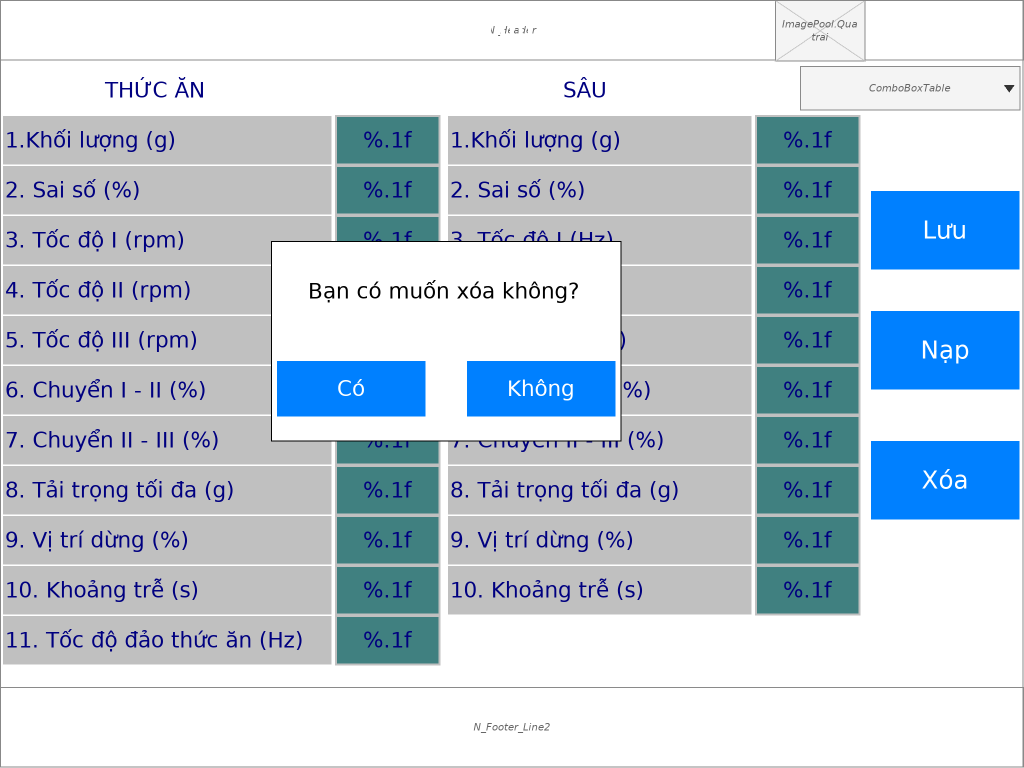
VISUALIZATION N_Recipe_Line2  // 1024x768
    Frame (0,687 1024x80)
        shows N_Footer_Line2()
    Frame (0,0 1024x60)
        shows N_Header()
    Textfield (353,5 400x50), "MÀN HÌNH LƯU THÔNG SỐ LINE 2"
    Textfield (80,75 150x30), "THỨC ĂN"
    Textfield (545,75 80x30), "SÂU"
    Rectangle (870,190 150x80), "Lưu"
        tap GVL_OF_VU.bRecSave[2]
        OnDialogClosed: execute { bSave2 := true; }
        OnMouseDown: write PRG_MainRecipe1_1.NameSave via VisuDialogs.Keypad
    Rectangle (870,440 150x80), "Xóa"
        tap GVL_OF_VU.bRecDelete[2]
        OnMouseClick: execute { GVL_OF_VU.bDeleteRecipe2 := true; }
    Rectangle (870,310 150x80), "Nạp"
        tap GVL_OF_VU.bRecLoad[2]
        OnMouseClick: execute { bLoad2 := true; }
    Group (447,115 305x500)
        Rectangle (0,0 305x50), "1.Khối lượng (g)"
        Rectangle (0,50 305x50), "2. Sai số (%)"
        Rectangle (0,100 305x50), "3. Tốc độ I (Hz)"
        Rectangle (0,150 305x50), "4. Tốc độ II (Hz)"
        Rectangle (0,250 305x50), "6. Chuyển I - II (%)"
        Rectangle (0,350 305x50), "8. Tải trọng tối đa (g)"
        Rectangle (0,200 305x50), "5. Tốc độ III (Hz)"
        Rectangle (0,300 305x50), "7. Chuyển II - III (%)"
        Rectangle (0,450 305x50), "10. Khoảng trễ (s)"
        Rectangle (0,400 305x50), "9. Vị trí dừng (%)"
    Textfield (755,115 105x50), "%.1f", text variable: PR_Line02.fDerisedWeight_Worm
    Textfield (755,165 105x50), "%.1f", text variable: PR_Line02.fDelta_Worm
    Textfield (755,215 105x50), "%.1f", text variable: PR_Line02.fFast_Speed_vibrating_funnel
    Textfield (755,265 105x50), "%.1f", text variable: PR_Line02.fSlow_Speed_vibrating_funnel_1
    Textfield (755,315 105x50), "%.1f", text variable: PR_Line02.fSlow_Speed_vibrating_funnel_2
    Textfield (755,365 105x50), "%.1f", text variable: PR_Line02.fChangeMode_Worm_1
    Textfield (755,415 105x50), "%.1f", text variable: PR_Line02.fChangeMode_Worm_2
        OnMouseDown: write GVL_OF_VU.fRecChangeII_IIIOfWorm[2] via VisuDialogs.Numpad
    Textfield (755,465 105x50), "%.1f", text variable: PR_Line02.fMaxWeight_Worm
    Textfield (755,515 105x50), "%.1f", text variable: PR_Line02.fPerStop_Worm
    Textfield (755,565 105x50), "%.1f", text variable: PR_Line02.fTimer_check_Worm
    Rectangle (2,115 330x50), "1.Khối lượng (g)"
    Rectangle (2,165 330x50), "2. Sai số (%)"
    Rectangle (2,215 330x50), "3. Tốc độ I (rpm)"
    Rectangle (2,265 330x50), "4. Tốc độ II (rpm)"
    Rectangle (2,365 330x50), "6. Chuyển I - II (%)"
    Rectangle (2,465 330x50), "8. Tải trọng tối đa (g)"
    Rectangle (2,315 330x50), "5. Tốc độ III (rpm)"
    Rectangle (2,415 330x50), "7. Chuyển II - III (%)"
    Rectangle (2,565 330x50), "10. Khoảng trễ (s)"
    Rectangle (2,515 330x50), "9. Vị trí dừng (%)"
    Rectangle (2,615 330x50), "11. Tốc độ đảo thức ăn (Hz)"
    Textfield (335,115 105x50), "%.1f", text variable: PR_Line02.fDerisedWeight_Food
    Textfield (335,165 105x50), "%.1f", text variable: PR_Line02.fDelta_Food
    Textfield (335,215 105x50), "%.1f", text variable: PR_Line02.fFast_Speed
    Textfield (335,265 105x50), "%.1f", text variable: PR_Line02.fSlow_Speed_1
    Textfield (335,315 105x50), "%.1f", text variable: PR_Line02.fSlow_Speed_2
    Textfield (335,365 105x50), "%.1f", text variable: PR_Line02.fChangeMode_Food_1
    Textfield (335,415 105x50), "%.1f", text variable: PR_Line02.fChangeMode_Food_2
    Textfield (335,465 105x50), "%.1f", text variable: PR_Line02.fMaxWeight_Food
    Textfield (335,515 105x50), "%.1f", text variable: PR_Line02.fPerStop_Food
    Textfield (335,565 105x50), "%.1f", text variable: PR_Line02.fTimer_Check_Food
    Textfield (335,615 105x50), "%.1f", text variable: PR_Line02.fSpeed_motor_mixer
    Image (775,0 90x61), image: ImagePool.Qua trai
        OnMouseClick: change screen: N_Recipe_Line1
    ComboBoxTable (800,66 220x44), variable: PRG_MainRecipe1_1.RecipeNameIdx, data array: PRG_MainRecipe1_1.RecipeList
        p3854506369: PRG_MainRecipe1_1.RecipeList[INDEX]
    GroupBox (271,241 350x200), invisible if: not GVL_OF_VU.bDeleteRecipe2, input disabled if: not GVL_OF_VU.bDeleteRecipe2
        Rectangle (0,0 350x200)
        Rectangle (5,119 150x57), "Có"
            OnMouseDown: execute { bDelete2 := true; }
            OnMouseUp: execute { GVL_OF_VU.bDeleteRecipe2 := FALSE; }
        Label (4,29 338x42), "Bạn có muốn xóa không?"
        Rectangle (195,119 150x57), "Không"
            OnMouseDown: execute { GVL_OF_VU.bDeleteRecipe2 := FALSE; }
END_VISUALIZATION

(* stored: Version 1.1.0.1, ProductVersion 3.1.4024.12
   Visu N_Recipe_Line2: Id {f6119dcf-be68-459a-b8f2-210d44f541db} *)
